// TIA Portal project "Projekt-Versionverwaltung1" (V20)

(* hardware
DEVICE "ET 200SP-Station_1"  ET 200SP-Station
   slot 0: "Baugruppenträger_0"  Rack  6ES5 710-8MAx1
   slot 0: "IO-Device_1"  IM 155-6 PN ST  6ES7 155-6AU00-0BN0  V3.3
   slot 127: "BA 2xRJ45"  BA 2xRJ45  6ES7 193-6AR00-0AA0  V0.0
      slot 1: "Port_1"  X1 P1R  6ES7 193-6AR00-0AA0  V0.0
      slot 2: "Port_2"  X1 P2R  6ES7 193-6AR00-0AA0  V0.0
DEVICE "S7-1500/ET200MP-Station_1"  S7-1500 station
   slot 0: "Profilschiene_0"  Rack  6ES7 590-1***0-0AA0
   slot 1: "PLC_1"  CPU 1515F-2 PN  6ES7 515-2FM01-0AB0  V2.9
      slot 3: "CPU-Display_1"  6ES7591-1BA00-0AA0
      slot 32768: "PROFINET-Schnittstelle_1"  X1
         slot 32769: "Port_1"  X1 P1
         slot 32770: "Port_2"  X1 P2
      slot 33024: "PROFINET-Schnittstelle_2"  X2
         slot 33025: "Port_1"  X2 P1
      slot 34817: "Virtual CP interface port_1"  Virtual CP interface port  Virtual CP interface port
   slot 2: "DI 16x24VDC HF_1"  DI 16x24VDC HF  6ES7 521-1BH00-0AB0  V2.2
   slot 3: "DQ 8x24VDC/2A HF_1"  DQ 8x24VDC/2A HF  6ES7 522-1BF00-0AB0  V2.2
DEVICE "HMI_1"  TP700 Comfort INOX PCT Portrait
   slot 0: "HMI_1"  TP700 Comfort INOX PCT PORTRAIT  6AV2 144-8GC20-0AA0  17.0.0.0
   slot 1: "HMI_RT_1"  TP700 Comfort INOX PCT PORTRAIT  6AV2 144-8GC20-0AA0  17.0.0.0
   slot 5: "HMI_1.IE_CP_1"  PROFINET Interface  17.0.0.0
      slot 1: "PROFINET Schnittstelle_1"  PROFINET Interface
         slot 1: "Port_1"  Port
         slot 2: "Port_2"  Port
   slot 7: "HMI_1.MPI/DP_CP_1"  MPI/DP Interface  17.0.0.0
*)

// ===== PLC "PLC_1"  CPU 1515F-2 PN =====

VAR_GLOBAL   // PLC tag table "Standard-Variablentabelle"
   "Tag_1" AT %Q0.3 : Bool;
END_VAR

VAR_GLOBAL   // PLC tag table "Eingänge"
   "Start_RLauf" AT %I0.0 : Bool;
   "Start-LLauf" AT %I0.1 : Bool;
   "StopTaste" AT %I0.2 : Bool;
END_VAR

VAR_GLOBAL   // PLC tag table "Ausgänge"
   "MRLauf" AT %Q0.0 : Bool;
   "MLLauf" AT %Q0.1 : Bool;
   "MLampe" AT %Q0.2 : Bool;
END_VAR

DATA_BLOCK "Main_Safety_RTG1_DB"   // DB1, F_DB
{ S7_Optimized_Access := 'TRUE' }
NAME : FUSI
VERSION : 0.1
// stored: InstanceOfName Main_Safety_RTG1
"Main_Safety_RTG1"
BEGIN
END_DATA_BLOCK

FUNCTION_BLOCK "Main_Safety_RTG1"   // FB1, F_FBD
{ S7_Optimized_Access := 'TRUE' }
BEGIN
END_FUNCTION_BLOCK

FUNCTION_BLOCK "Baustein_KOP"   // FB2, LAD
{ S7_Optimized_Access := 'TRUE' }
VERSION : 0.1
BEGIN

REGION Network 1: Rechtslauf
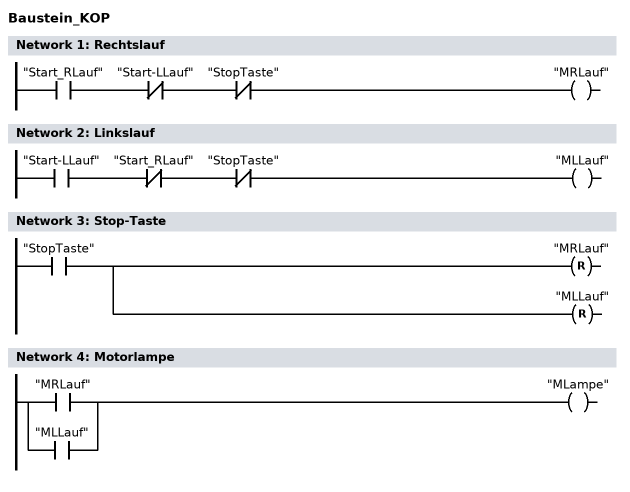
   RUNG wire#powerrail
      Contact( "Start_RLauf" )
      I_Contact( "Start-LLauf" )
      I_Contact( "StopTaste" )
      Coil( "MRLauf" )
   END_RUNG
   // the same network as SCL:
   "MRLauf" := "Start_RLauf" AND NOT "Start-LLauf" AND NOT "StopTaste";
END_REGION

REGION Network 2: Linkslauf
   RUNG wire#powerrail
      Contact( "Start-LLauf" )
      I_Contact( "Start_RLauf" )
      I_Contact( "StopTaste" )
      Coil( "MLLauf" )
   END_RUNG
   // the same network as SCL:
   "MLLauf" := "Start-LLauf" AND NOT "Start_RLauf" AND NOT "StopTaste";
END_REGION

REGION Network 3: Stop-Taste
   RUNG wire#powerrail
      Contact( "StopTaste" )
      wire#w1
      R_Coil( "MRLauf" )
   END_RUNG
   RUNG wire#w1
      R_Coil( "MLLauf" )
   END_RUNG
   // the same network as SCL:
   IF "StopTaste" THEN
       "MRLauf" := FALSE;
       "MLLauf" := FALSE;
   END_IF;
END_REGION

REGION Network 4: Motorlampe
   RUNG wire#powerrail
      Contact( "MRLauf" )
      wire#w1
      Coil( "MLampe" )
   END_RUNG
   RUNG wire#powerrail
      Contact( "MLLauf" )
   END_RUNG wire#w1
   // the same network as SCL:
   "MLampe" := "MRLauf" OR "MLLauf";
END_REGION
END_FUNCTION_BLOCK

FUNCTION_BLOCK "Baustein_SCL"   // FB3, SCL
{ S7_Optimized_Access := 'TRUE' }
VERSION : 0.1
BEGIN
   // Motorsteuerung Rechts-/Linkslauf

   IF "StopTaste"  THEN             // Stop-Taste
       "MRLauf" := FALSE;
       "MLLauf" := FALSE;
   ELSE

       IF "Start_RLauf" AND NOT "MLLauf" THEN
       "MRLauf" := TRUE;
       END_IF;

       // Linkslauf
       IF "Start-LLauf"AND NOT "MRLauf"  THEN
           "MLLauf" := TRUE;
       END_IF;
   END_IF;

   // Rückmeldung: Motor läuft
   "MLampe" := "MLLauf" OR "MRLauf";
END_FUNCTION_BLOCK

FUNCTION "Baustein_AWL" : Void   // FC1, STL
{ S7_Optimized_Access := 'TRUE' }
VERSION : 0.1
BEGIN

REGION Network 1: Rechtslauf
         A     "Start_RLauf";
         AN    "MLLauf";
         S     "MRLauf";
END_REGION

REGION Network 2: Linkslauf
         A     "Start-LLauf";
         AN    "MRLauf";
         S     "MLLauf";
END_REGION

REGION Network 3: Stop Taste
         A     "StopTaste";
         R     "MRLauf";
         R     "MLLauf";
END_REGION

REGION Network 4: Motor Lampe
         A     "MRLauf";
         O     "MLLauf";
         =     "MLampe";
END_REGION
END_FUNCTION

FUNCTION "Baustein_FUP" : Void   // FC2, FBD
{ S7_Optimized_Access := 'TRUE' }
VERSION : 0.1
BEGIN

REGION Network 1: Rechtslauf starten
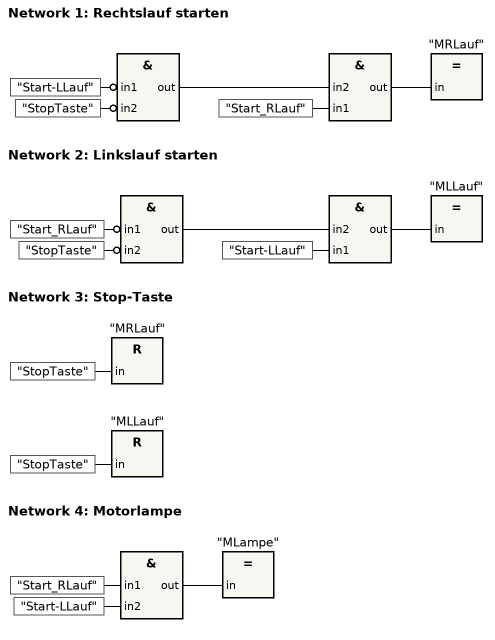
   "MRLauf" := NOT "Start-LLauf" AND NOT "StopTaste" AND "Start_RLauf";
END_REGION

REGION Network 2: Linkslauf starten
   "MLLauf" := NOT "Start_RLauf" AND NOT "StopTaste" AND "Start-LLauf";
END_REGION

REGION Network 3: Stop-Taste
   IF "StopTaste" THEN
       "MRLauf" := FALSE;
       "MLLauf" := FALSE;
   END_IF;
END_REGION

REGION Network 4: Motorlampe
   "MLampe" := "Start_RLauf" AND "Start-LLauf";
END_REGION
END_FUNCTION

ORGANIZATION_BLOCK "Main"   // OB1, LAD, ProgramCycle
TITLE = "Main Program Sweep (Cycle)"
{ S7_Optimized_Access := 'TRUE' }
VERSION : 0.1
   VAR_INPUT
      Initial_Call : Bool;   // Initial call of this OB
      Remanence : Bool;   // =True, if remanent data are available
   END_VAR
BEGIN
END_ORGANIZATION_BLOCK